// Get the distance to travel from startPos to stopPos
FUNCTION DistToTravel : LREAL
VAR_INPUT
    startPos : LREAL;
    stopPos  : LREAL;
END_VAR
VAR
END_VAR

IF startPos > stopPos THEN
    DistToTravel := stopPos - startPos + CONST.MAX_TRACK_LENGTH;
ELSE
    DistToTravel := stopPos - startPos;
END_IF

END_FUNCTION

(* stored: Version 1.1.0.1, ProductVersion 3.1.4024.12
   POU DistToTravel: Id {55aa1e87-f348-47c2-aeed-49f339215e5e}, SpecialFunc None *)
